      ######################## affichage_POPUP #####################################
      sync()
      num_soud = to_str(num)
      popup1 = "popup Config. : " + type_soud + " n°" + num_soud + " : placer " + etape_soud + " & Valider"             #on ouvre un popup
      socket_open("127.0.0.1", 29999, "internal") # open internal socket
      socket_send_line(popup1, "internal")     #Affichage message
      socket_send_byte(10, "internal")
      sync()
  end
  #-

  def popUp_tropSoudures():
      close_popup()
      popUp_tropSoudures = "Ajout impossible, deja 10 soudures de ce type"
      socket_open("127.0.0.1",29999,"internal") # open internal socket
      socket_send_line(popUp_tropSoudures,"internal")     #Affichage message
      socket_send_byte(10,"internal")
  end
  #-
  $ 41 "Mouvements soudures"
  $ 42 "Script: fcts_balayage.script"
  def fct_determineAxeBalayage(p_start,p_stop):

      global  diff_x = norm(p_start[0]-p_stop[0])
      global  diff_y = norm(p_start[1]-p_stop[1])
      global  diff_z = norm(p_start[2]-p_stop[2])

      global offset_x =  0
      global offset_y =  0
      global offset_z = 0

      local tolerance = 0.02



      if ( (diff_z >0.05) ):
          offset_z = 1
      end

      if ( (diff_x >tolerance) or (offset_z == 1)):
          offset_y = 1
      end

      if ( (diff_y >tolerance) or (offset_z == 1)):
          offset_x = 1
      end

  end

  def fct_set_offset():

      if (offset_x == 1):
          offset[0] = sin((i/cycle_duration)*2.0*pi) * amplitude
      end

      if (offset_y == 1):
          offset[1] = sin((i/cycle_duration)*2.0*pi) * amplitude
      end

  end

  thread runBalayage():
    while (True):
        global ctrl_frequency=350.0
        global weave_frequency=1.2
        global amplitude=0.003
        global cycle_duration=(ctrl_frequency / weave_frequency)
        global pi=3.14159
        global offset=[0.0, 0.0, 0.0, 0.0, 0.0, 0.0]
        global i=0
        path_offset_enable()
        global alpha=0.1
        path_offset_set_alpha_filter(alpha)

        while (True):
          fct_set_offset()
          path_offset_set(offset, 2)
          global i=i+1
          sync()
        end
      end

  end

  def fct_activerBalayage(p_start, p_stop,amplitude, frequence):

      fct_determineAxeBalayage(p_start,p_stop)
      amplitude_thr = amplitude
      frequence_thr = frequence
      global thr_runBalayage = run runBalayage()

  end

  def fct_desactiverBalayage():

      kill thr_runBalayage

  end

  def fct_demande_amplitude():

      amplitude = request_integer_from_primary_client("amplitude du balayage en mm :")
      while (amplitude <=0):
          amplitude = request_integer_from_primary_client("amplitude du balayage en mm :")
      end

      amplitude = amplitude/1000

      return amplitude

  end


  def fct_demande_frequence():

      frequence = request_float_from_primary_client("frequence du balayage en Hz :")
      while (frequence <=0):
          frequence = request_float_from_primary_client("frequence du balayage en Hz :")
      end

      return frequence

  end
  $ 43 "Script: fcts_ralentir_fin_ligne.script"
  def fct_calcul_point_inter(p_debut,p_fin):

      local p_inter = p_fin

      local poucentage = 0.95
      local inc = 0
      local vecteur_global = p[0,0,0,0,0,0]
      local vecteur_reduit = p[0,0,0,0,0,0]

      while (inc < 6):   #a valider avec d'autres tests (peut etre faire une moyenne)
          vecteur_global[inc] = p_fin[inc] - p_debut[inc]
          vecteur_reduit[inc] = vecteur_global[inc]*poucentage
          p_inter[inc] = p_debut[inc] + vecteur_reduit[inc]
          inc = inc +1
      end

      return p_inter
    end


  $ 44 "General"
  $ 45 "Script: diverses.script"
  def attente_carters_ouverts():
      global debug = 2
      # vérifier que les carter sont ouverts,
      # sinon attendre en faisant clignoter les leds

      while ((get_configurable_digital_in(add_SecuGaucheOk) == True) or (get_configurable_digital_in(add_SecuDroiteOK) == True)):

          sync()
          # 94 "'clingottement pour signifier qu'il y  un defaut sur un des carters '"
          set_standard_digital_out(add_Dcy_Voyant, False)
          set_configurable_digital_out(add_Led_Arret, False)
          sleep(0.5)
          set_standard_digital_out(add_Dcy_Voyant, True)
          set_configurable_digital_out(add_Led_Arret, True)
          sleep(0.5)
          sync()
      end

      #carter OK, RAZ des sorties
      set_standard_digital_out(add_Dcy_Voyant, False)
      set_configurable_digital_out(add_Led_Arret, False)
      sleep(2)
      sync()

      global debug = 3

  end
  #-

  def deplacement_depart_init():

      global angle_base = get_actual_joint_positions ()
      if (angle_base[0] <= 0.7):
          if (angle_base[0] >= 1.6):
              # 116 "Départ"        A CHANGER PAR UNE POSTION ENREGISTREE
              movej(pose_depart, a = accelerationHorsSoudure, v = vitesseHorsSoudure)
          else:
              if (angle_base[0] > 1.6):
                  movej(Point_init_D, a = accelerationHorsSoudure, v = vitesseHorsSoudure)
                  movej(Point_avt_initD, a = accelerationHorsSoudure, v = vitesseHorsSoudure)
              else:
                  if (angle_base[0] < 0.7):
                      movej(Point_init_G, a = accelerationHorsSoudure, v = vitesseHorsSoudure)
                  end
              end
          end
      else:
          # 124 "SinonSi angle_base[0]>1.6"
          if (angle_base[0] > 1.6):

              movej(Point_init_D, a = accelerationHorsSoudure, v = vitesseHorsSoudure)
              movej(Point_avt_initD, a = accelerationHorsSoudure, v = vitesseHorsSoudure)
          else:
              if (angle_base[0] < 0.7):
                  movej(Point_init_G, a = accelerationHorsSoudure, v = vitesseHorsSoudure)
              end
          end
      end
      # 131 "Départ"             A CHANGER PAR UNE POSTION ENREGISTREE
      movej(pose_depart, a = accelerationHorsSoudure, v = vitesseHorsSoudure)
      #global angle_base= get_actual_joint_positions ()
      sync()
  end
  #-

  def mode_configuration():
      #nouveau

      if ((config_g == 1) and (config_d == 1)):
          pop_up_config_g_et_d()
      elif ((config_g == 1) and (config_d == 0)):
          pop_up_config_g()
      elif ((config_g == 0) and (config_d == 1)):
          pop_up_config_d()
      elif ((config_g == 0) and (config_d == 0)):
          pop_up_config()
      end

      while ((get_configurable_digital_in(add_ModeExe) == False  ) and (get_standard_digital_in(add_bp_ConfigReglage) == False  )):
          thread Thread_while_145():
              while (True):  # faire clignoter les voyants des tables, pour informer de l'attente d'une action
                  set_standard_digital_out(add_VoyantTableDroite, True)
                  set_standard_digital_out(add_VoyantTableGauche, False)
                  sleep(0.5)
                  set_standard_digital_out(add_VoyantTableDroite, False)
                  set_standard_digital_out(add_VoyantTableGauche, True)
                  sleep(0.5)
                  sync()
              end
          end
          if (get_standard_digital_in(adresse_bp_d) == False and get_standard_digital_in(adresse_bp_g) == False and get_configurable_digital_in(add_ModeExe) == False and get_standard_digital_in(add_bp_ConfigReglage) == False):
              global thread_handler_145 = run Thread_while_145()
              while (get_standard_digital_in(adresse_bp_d) == False and get_standard_digital_in(adresse_bp_g) == False and get_configurable_digital_in(add_ModeExe) == False and get_standard_digital_in(add_bp_ConfigReglage) == False):
                  sync()
              end
              kill thread_handler_145
          end
          if (get_standard_digital_in(adresse_bp_g) == True): #table gauche
              set_standard_digital_out(add_VoyantTableGauche, True)
              set_standard_digital_out(add_VoyantTableDroite, False)
              movej(Point_init_G, a = accelerationHorsSoudure, v = vitesseHorsSoudure, r = 0.006)
              movej(Point_Attente_G, a = accelerationHorsSoudure, v = vitesseHorsSoudure, r = 0.006)
              movej(Point_config_g, a = accelerationHorsSoudure, v = vitesseHorsSoudure)
              global led_cobot = 1
              fun_config_g()
              global led_cobot = 0
              fun_valid_config_g()
              movej(Point_Attente_G, a = accelerationHorsSoudure, v = vitesseHorsSoudure, r = 0.006)
              movej(Point_init_G, a = accelerationHorsSoudure, v = vitesseHorsSoudure, r = 0.006)
              # 170 "Départ"         A CHANGER PAR UNE POSTION ENREGISTREE
              movej(pose_depart, a = accelerationHorsSoudure, v = vitesseHorsSoudure)
          end

          if (get_standard_digital_in(adresse_bp_d) == True): #table droite
              set_standard_digital_out(add_VoyantTableDroite, True)
              set_standard_digital_out(add_VoyantTableGauche, False)
              movej(Point_avt_initD, a = accelerationHorsSoudure, v = vitesseHorsSoudure, r = 0.006)
              movej(Point_init_D, a = accelerationHorsSoudure, v = vitesseHorsSoudure)
              movej(Point_Attente_D, a = accelerationHorsSoudure, v = vitesseHorsSoudure, r = 0.006)
              movej(Point_config_d, a = accelerationHorsSoudure, v = vitesseHorsSoudure)
              global led_cobot = 1
              fun_config_d()
              global led_cobot = 0
              fun_valid_config_d()
              movej(Point_Attente_D, a = accelerationHorsSoudure, v = vitesseHorsSoudure, r = 0.006)
              movej(Point_init_D, a = accelerationHorsSoudure, v = vitesseHorsSoudure, r = 0.006)
              movej(Point_avt_initD, a = accelerationHorsSoudure, v = vitesseHorsSoudure, r = 0.006)
              # 190 "Départ"         A CHANGER PAR UNE POSTION ENREGISTREE
              movej(pose_depart, a = accelerationHorsSoudure, v = vitesseHorsSoudure)
          end
      end

      sync()
  end
  #-

  def mode_Reglage():
      #Pas à Pas
      if ((config_g == 1) and (config_d == 1)):
          pop_up_reg_gd()
          global boucle = 1
      elif ((config_g == 1) and (config_d == 0)):
          pop_up_reg_gd()
          global boucle = 1
      elif ((config_g == 0) and (config_d == 1)):
          pop_up_reg_d()
          global boucle = 1
      else:
          close_popup()
          while (get_standard_digital_in(add_bp_ConfigReglage) == True):
              popup("Aucune configuration n'est actuellement detectée.", "Erreur", False, True, blocking = True)
          end
      end



      global boucle = 1
      while ((get_configurable_digital_in(add_ModeExe) == False  ) and (boucle == 1) and (get_standard_digital_in(add_bp_ConfigReglage) == True  )):
          thread Thread_while_208():
              while (True):
                  if (config_g == 1):
                      set_standard_digital_out(add_VoyantTableGauche, True)
                  end
                  if (config_d == 1):
                      set_standard_digital_out(add_VoyantTableDroite, True)
                  end
                  sleep(0.5)
                  set_standard_digital_out(add_VoyantTableGauche, False)
                  set_standard_digital_out(add_VoyantTableDroite, False)
                  sleep(0.5)
              end
          end
          if (get_standard_digital_in(adresse_bp_d) == False and get_standard_digital_in(adresse_bp_g) == False and get_configurable_digital_in(add_ModeExe) == False and get_standard_digital_in(add_bp_ConfigReglage) == True):
              global thread_handler_208 = run Thread_while_208()
              while (get_standard_digital_in(adresse_bp_d) == False and get_standard_digital_in(adresse_bp_g) == False and get_configurable_digital_in(add_ModeExe) == False and get_standard_digital_in(add_bp_ConfigReglage) == True):
                  sync()
              end
              kill thread_handler_208
          end
          if (get_standard_digital_in(adresse_bp_g) == True): #table gauche
              global safe_mode = 1
              set_standard_digital_out(add_VoyantTableGauche, True)
              set_standard_digital_out(add_VoyantTableDroite, False)
              movej(Point_init_G, a = accelerationHorsSoudure, v = vitesseHorsSoudure, r = 0.006)
              movej(Point_Attente_G, a = accelerationHorsSoudure, v = vitesseHorsSoudure, r = 0.006)
              movej(pose_inter_g, a = accelerationHorsSoudure, v = vitesseHorsSoudure)
              global led_cobot = 1
              fun_Pas_A_Pas_g()
              global led_cobot = 0
              global safe_mode = 0
              global boucle = 0
          end
          if (get_standard_digital_in(adresse_bp_d) == True): #table droite
              global safe_mode = 1
              set_standard_digital_out(add_VoyantTableDroite, True)
              set_standard_digital_out(add_VoyantTableGauche, False)
              movej(Point_avt_initD, a = accelerationHorsSoudure, v = vitesseHorsSoudure, r = 0.006)
              movej(Point_init_D, a = accelerationHorsSoudure, v = vitesseHorsSoudure, r = 0.006)
              movej(pose_inter_d, a = accelerationHorsSoudure, v = vitesseHorsSoudure)
              global led_cobot = 1
              fun_Pas_A_Pas_d()
              global led_cobot = 0
              global safe_mode = 0
              global boucle = 0
          end
      end

      sync()
  end
  #-

  def mode_Execution():

      if ((config_g == 1) and (config_d == 1)):
          pop_up_exe()
          global boucle = 1
      elif ((config_g == 1) and (config_d == 0)):
          pop_up_exe_g()
          global boucle = 1
      elif ((config_g == 0) and (config_d == 1)):
          pop_up_exe_d()
          global boucle = 1
      else:
          close_popup()
          while (get_configurable_digital_in(add_ModeExe) == True):
              popup("Aucune programmation n'est actuellement detectée, veillez à programmer une pièce avant de vouloir l'éxécuter.", "Erreur", False, True, blocking = True)
          end
      end

      while (( get_configurable_digital_in(add_ModeExe) == True  ) and (boucle == 1)):
          thread Thread_while_259():
              while (True):
                  if (config_g == 1):
                      set_standard_digital_out(add_VoyantTableGauche, True)
                  end
                  if (config_d == 1):
                      set_standard_digital_out(add_VoyantTableDroite, True)
                  end
                  sleep(0.5)
                  set_standard_digital_out(add_VoyantTableGauche, False)
                  set_standard_digital_out(add_VoyantTableDroite, False)
                  sleep(0.5)
              end
          end

          if (get_standard_digital_in(adresse_bp_d) == False and get_standard_digital_in(adresse_bp_g) == False and get_configurable_digital_in(add_ModeExe) == True):
              global thread_handler_259 = run Thread_while_259()
              while (get_standard_digital_in(adresse_bp_d) == False and get_standard_digital_in(adresse_bp_g) == False and get_configurable_digital_in(add_ModeExe) == True):
                  sync()
              end
              kill thread_handler_259
          end

          if ((get_standard_digital_in(adresse_bp_g) == True  ) and (config_g == True  )): #table de gauche
              pop_up_deb_exe_g()
              global boucle_g = 1
              while (boucle_g == 1):  #Boucler une fois, tant que la soudure n'est pas finie
                  set_configurable_digital_out(add_CmdCarterBit1, True)#commande la fermeture du carter

                  set_standard_digital_out(add_VoyantTableGauche, True) #commande des voyants
                  set_standard_digital_out(add_VoyantTableDroite, False)
                  sleep(0.25)
                  set_standard_digital_out(add_VoyantTableGauche, False)
                  sleep(0.25)

                  if (get_configurable_digital_in(add_SecuGaucheOk) == False): #si les carter ne sont pas en position : voyant et attente
                      set_standard_digital_out(add_VoyantTableGauche, True)
                      while (get_configurable_digital_in(add_SecuGaucheOk) == False):
                          sync()
                      end
                  end

                  if (get_configurable_digital_in(add_SecuGaucheOk) == True): # attente de la confirmation de la position du carter -> début soudure
                      global secu_g = 1
                      set_standard_digital_out(add_VoyantTableGauche, True)
                      movej(Point_init_G, a = accelerationHorsSoudure, v = vitesseHorsSoudure, r = 0.006)
                      fun_execution_g()
                      movej(Point_Attente_G, a = accelerationHorsSoudure, v = vitesseHorsSoudure, r = 0.006)
                      movej(Point_init_G, a = accelerationHorsSoudure, v = vitesseHorsSoudure, r = 0.006)
                      # 294 "Départ"         A CHANGER PAR UNE POSTION ENREGISTREE
                      movej(pose_depart, a = accelerationHorsSoudure, v = vitesseHorsSoudure)
                      set_configurable_digital_out(add_CmdCarterBit1, False)
                      global secu_g = 0
                      global boucle_g = 0
                  end
              end
              global boucle = 0
          else:
              if ((get_standard_digital_in(adresse_bp_g) == True  ) and (config_g == False  )): # si la table n'est pas enregistrée comme configurée
                  close_popup()
                  popup("Aucune programmation n'est actuellement detectée sur la table gauche, veillez à programmer une pièce avant de vouloir l'éxécuter.", "Erreur", False, True, blocking = True)
                  global boucle = 0
              end
          end
          if ((get_standard_digital_in(adresse_bp_d) == True  ) and (config_d == True  )):  #table de droite
              global boucle_d = 1
              pop_up_deb_exe_d()
              while (boucle_d == 1):  #Boucler une fois, tant que la soudure n'est pas finie
                  set_configurable_digital_out(add_CmdCarterBit2, True) #commande la fermeture du carter

                  set_standard_digital_out(add_VoyantTableGauche, False)#commande des voyants
                  set_standard_digital_out(add_VoyantTableDroite, True)
                  sleep(0.25)
                  set_standard_digital_out(add_VoyantTableDroite, False)
                  sleep(0.25)

                  if (get_configurable_digital_in(add_SecuDroiteOK) == False): #si les carter ne sont pas en position : voyant et attente
                      set_standard_digital_out(add_VoyantTableDroite, True)
                      while (get_configurable_digital_in(add_SecuDroiteOK) == False):
                          sync()
                      end
                  end

                  if (get_configurable_digital_in(add_SecuDroiteOK) == True):# attente de la confirmation de la position du carter -> début soudure
                      global secu_d = 1
                      set_standard_digital_out(add_VoyantTableDroite, True)
                      movej(Point_avt_initD, a = accelerationHorsSoudure, v = vitesseHorsSoudure)
                      fun_execution_d()
                      set_configurable_digital_out(add_CmdCarterBit2, False)
                      global secu_d = 0
                      global boucle_d = 0
                  end
              end
              global boucle = 0
          else:
              if ((get_standard_digital_in(adresse_bp_d) == True  ) and (config_d == False  )): # si la table n'est pas enregistrée comme configurée
                  close_popup()
                  popup("Aucune programmation n'est actuellement detectée sur la table droite, veillez à programmer une pièce avant de vouloir l'éxécuter.", "Erreur", False, True, blocking = True)
                  global boucle = 0
              end
          end
      end
      sync()
  end
  #-
  $ 46 "Script: general.script"
  def General():

      while (True):

          global debug = 1
          #INTIALISATION
          safe_mode = 0
          set_configurable_digital_out(add_CmdCarterBit1, False) #stop commande carter
          set_configurable_digital_out(add_CmdCarterBit2, False)

          attente_carters_ouverts() #éviter un contact avec le bras

          deplacement_depart_init() #premier déplacement à gérer en focntion de la position réel du robot lors de l'init

          # TEST DES MODES :
          # lecture de la postion des Bps
          if ((get_configurable_digital_in(add_ModeExe) == False) and (get_standard_digital_in(add_bp_ConfigReglage) == False)):
              mode_configuration()#l 55-> 127
          elif ((get_configurable_digital_in(add_ModeExe) == False) and (get_standard_digital_in(add_bp_ConfigReglage) == True  )):
              mode_Reglage() #l 127 -> 199
          elif (get_configurable_digital_in(add_ModeExe) == True):
              mode_Execution() #
          else:
              #faire erreur
          end
      end

  end
  $ 76 "Thread_1"
  thread Thread_1():
    while (True):
      $ 77 "Test_Ordre_Marche"
      $ 78 "If Test_Ordre_Mar≟ True "
      if (Test_Ordre_Mar ==   True  ):
        $ 79 "If config_d ≟ 1  or  config_g ≟ 1"
        if (config_d  ==  1   or   config_g  ==  1):
          $ 80 "Set Ordre_Marche=On"
          set_standard_digital_out(0, True)
          $ 81 "Wait: 0.5"
          sleep(0.5)
          $ 82 "If Reponse_Ordre≟ False "
          if (get_standard_digital_in(4) ==   False  ):
            $ 83 "'Si aucune reponse n'a etait recue, arret du programme'"
            # 'Si aucune reponse n'a etait recue, arret du programme'
            $ 84 "close_popup()"
            close_popup()
            $ 85 "Popup: Defaut : L'Ordre marche a ete coupe ( le poste est peu-etre eteint ) "
            popup("Defaut : L'Ordre marche a ete coupe ( le poste est peu-etre eteint ) ", "Error", False, True, blocking=False)
            halt
          end
          $ 86 "Test_Ordre_Mar≔ False "
          global Test_Ordre_Mar=  False
          $ 87 "sync()"
          sync()
        end
      end
      $ 88 "Erreur ordre marche pendant utilisation"
      $ 89 "If Arc_On≟ True   and Reponse_Arc≟ True  and Reponse_Ordre≟ False "
      if (get_standard_digital_out(1) ==   True     and  get_standard_digital_in(5) ==   True    and  get_standard_digital_in(4) ==   False  ):
        $ 90 "'Test pour savoir si ordre marche a ete coupe pendant utilisation'"
        # 'Test pour savoir si ordre marche a ete coupe pendant utilisation'
        $ 91 "close_popup()"
        close_popup()
        $ 92 "Popup: Defaut : Mise sous puissance coupee pendant la trajectoire"
        popup("Defaut : Mise sous puissance coupee pendant la trajectoire", "Error", False, True, blocking=False)
        halt
      end
      $ 93 "sync()"
      sync()
    end
  end
  threadId_Thread_1 = run Thread_1()
  $ 94 "Thread_2"
  thread Thread_2():
    while (True):
      $ 95 "mode_soudure"
      $ 96 "If Mode_soudure ≟  True "
      if (get_configurable_digital_in(3)  ==    True  ):
        $ 97 "If Mode_soudure≟ True  and soudure_on ≟ True "
        if (get_configurable_digital_in(3) ==   True    and  soudure_on  ==   True  ):
          $ 98 "fin_soud≔0"
          global fin_soud=0
          $ 99 "Test_Ordre_Mar≔ True "
          global Test_Ordre_Mar=  True
          $ 100 "Test_Job≔ True "
          global Test_Job=  True
          $ 101 "Wait Test_Ordre_Mar≟ False "
          while (not(Test_Ordre_Mar ==   False  )):
            sync()
          end
          $ 102 "Wait Test_Job≟ False "
          while (not(Test_Job ==   False  )):
            sync()
          end
          $ 103 "Set Arc_On=On"
          set_standard_digital_out(1, True)
          $ 104 "Test_Gaz≔ True "
          global Test_Gaz=  True
          $ 105 "'Test_Gaz permet de faire un appel dans le thread pour tester l'arriver gaz'"
          # 'Test_Gaz permet de faire un appel dans le thread pour tester l'arriver gaz'
          $ 106 "Wait Valide_Gaz≟ True "
          while (not(Valide_Gaz ==   True  )):
            sync()
          end
          $ 107 "'Valide_Gaz permet  de connaitre quand le traitement de l'arriver gaz est terminer ans le thread.'"
          # 'Valide_Gaz permet  de connaitre quand le traitement de l'arriver gaz est terminer ans le thread.'
        else:
          $ 108 "ElseIf Mode_soudure ≟ True  and soudure_on ≟ False "
          if (get_configurable_digital_in(3)  ==   True    and  soudure_on  ==   False  ):
            $ 109 "'Attente post debit gaz'"
            # 'Attente post debit gaz'
            $ 110 "Set Arc_On=Off"
            set_standard_digital_out(1, False)
            $ 111 "Test_Gaz≔ False "
            global Test_Gaz=  False
            $ 112 "Loop Reponse_Arc ≟ 1"
            while (get_standard_digital_in(5)  ==  1):
              $ 113 "fin_soud≔0"
              global fin_soud=0
              $ 114 "sync()"
              sync()
            end
            $ 115 "fin_soud≔1"
            global fin_soud=1
          end
        end
      end
      $ 116 "sync()"
      sync()
    end
  end
  threadId_Thread_2 = run Thread_2()
  $ 117 "Thread_3"
  thread Thread_3():
    while (True):
      $ 118 "led_cobot_2"
      $ 119 "If led_cobot ≟ True "
      if (led_cobot  ==   True  ):
        $ 120 "If valider_bp_co ≟ True "
        if (get_tool_digital_in(0)  ==   True  ):
          $ 121 "Loop 3 times"
          Loop_4 = 0
          while (Loop_4 < 3):
            $ 122 "Set TO[1]=On"
            set_tool_digital_out(1, True)
            $ 123 "Wait: 0.25"
            sleep(0.25)
            $ 124 "Set TO[1]=Off"
            set_tool_digital_out(1, False)
            $ 125 "Wait: 0.25"
            sleep(0.25)
            $ 126 "sync()"
            sync()
            Loop_4 = Loop_4 + 1
          end
        end
        $ 127 "sync()"
        sync()
      end
      $ 128 "sync()"
      sync()
      $ 129 "sync()"
      sync()
    end
  end
  threadId_Thread_3 = run Thread_3()
  $ 130 "Thread_4"
  thread Thread_4():
    while (True):
      $ 131 "led_cobot"
      $ 132 "If led_cobot ≟ True "
      if (led_cobot  ==   True  ):
        $ 133 "Loop led_cobot ≟  True "
        while (led_cobot  ==    True  ):
          $ 134 "Set TO[0]=On"
          set_tool_digital_out(0, True)
          $ 135 "Wait: 0.5"
          sleep(0.5)
          $ 136 "Set TO[0]=Off"
          set_tool_digital_out(0, False)
          $ 137 "Wait: 0.5"
          sleep(0.5)
          $ 138 "sync()"
          sync()
        end
        $ 139 "sync()"
        sync()
      else:
        $ 140 "Else" "noBreak"
        $ 141 "Set TO[0]=Off"
        set_tool_digital_out(0, False)
        $ 142 "Set TO[1]=Off"
        set_tool_digital_out(1, False)
      end
      $ 143 "sync()"
      sync()
    end
  end
  threadId_Thread_4 = run Thread_4()
  $ 144 "Thread_5"
  thread Thread_5():
    while (True):
      $ 145 "Test_Arc_On"
      $ 146 "Erreur gaz pendant utilisation"
      $ 147 "Timer_gaz"
      $ 148 "If Test_Gaz≟ True "
      if (Test_Gaz ==   True  ):
        $ 149 "Wait: 1.0"
        sleep(1.0)
        $ 150 "Loop Reponse_Arc≟ False  and Arc_On≟ True "
        thread Thread_while_150():
          while (True):
            $ 151 "'La boucle permet d'activer le timer et tester deux condition pour les Defaults'"
            # 'La boucle permet d'activer le timer et tester deux condition pour les Defaults'
            $ 152 "timer_ret_gaz: Start"
            timer_ret_gaz_is_counting = True
            $ 153 "If timer_ret_gaz>0.5"
            global thread_flag_153=0
            thread Thread_if_153():
              $ 154 "'Le timer permet de realiser une attente '"
              # 'Le timer permet de realiser une attente '
              $ 155 "close_popup()"
              close_popup()
              $ 156 "Popup: Defaut : Pas de retour flux, stabilisation gaz"
              popup("Defaut : Pas de retour flux, stabilisation gaz", "Error", False, True, blocking=False)
              halt
              $ 157 "sync()"
              sync()
              thread_flag_153 = 1
            end
            if (timer_ret_gaz>0.5):
              global thread_handler_153=run Thread_if_153()
              while (thread_flag_153 == 0):
                if not(timer_ret_gaz>0.5):
                  kill thread_handler_153
                  thread_flag_153 = 2
                else:
                  sync()
                end
              end
            else:
              thread_flag_153 = 2
            end
            if (thread_flag_153 == 2):
              $ 158 "ElseIf Reponse_Ordre≟ False "
              if (get_standard_digital_in(4) ==   False  ):
                $ 159 "'Cette condition nous permet de pouvoir tout couper ordre marche pendant la boucle.'"
                # 'Cette condition nous permet de pouvoir tout couper ordre marche pendant la boucle.'
                $ 160 "close_popup()"
                close_popup()
                $ 161 "Popup: Defaut : Perte retour de signal, mise sous puissance generateur"
                popup("Defaut : Perte retour de signal, mise sous puissance generateur", "Error", False, True, blocking=False)
                halt
                $ 162 "sync()"
                sync()
              end
            end
          end
        end
        if (get_standard_digital_in(5) ==   False    and  get_standard_digital_out(1) ==   True  ):
          global thread_handler_150=run Thread_while_150()
          while (get_standard_digital_in(5) ==   False    and  get_standard_digital_out(1) ==   True  ):
            sync()
          end
          kill thread_handler_150
        end
        $ 163 "Valide_Gaz≔ True "
        global Valide_Gaz=  True
        $ 164 "timer_ret_gaz: Reset"
        timer_ret_gaz = 0
        $ 165 "sync()"
        sync()
      end
      $ 166 "sync()"
      sync()
    end
  end
  threadId_Thread_5 = run Thread_5()
  $ 175 "Thread_7"
  thread Thread_7():
    while (True):
      $ 176 "secu"
      $ 177 "If SecuGaucheOk ≟  False  and secu_g ≟ 1"
      if (get_configurable_digital_in(4)  ==    False    and  secu_g  ==  1):
        $ 178 "close_popup()"
        close_popup()
        $ 179 "Popup: ATTENTION : Defaut carter !"
        popup("ATTENTION : Defaut carter !", "Error", False, True, blocking=False)
        halt
      else:
        $ 180 "ElseIf SecuDroiteOk ≟ False  and secu_d ≟ 1"
        if (get_configurable_digital_in(5)  ==   False    and  secu_d  ==  1):
          $ 181 "close_popup()"
          close_popup()
          $ 182 "Popup: ATTENTION : Defaut carter !"
          popup("ATTENTION : Defaut carter !", "Error", False, True, blocking=False)
          halt
        end
      end
      $ 183 "sync()"
      sync()
    end
  end
  threadId_Thread_7 = run Thread_7()
  $ 184 "Thread_8"
  thread Thread_8():
    while (True):
      $ 185 "bloq_soud_arret"
      $ 186 "If Mode_soudure≟ False  and Test_Gaz ≟ True "
      if (get_configurable_digital_in(3) ==   False    and  Test_Gaz  ==   True  ):
        $ 187 "close_popup()"
        close_popup()
        $ 188 "Popup: Defaut : L'ordre de soudure a ete coupe pendant l'utilisation."
        popup("Defaut : L'ordre de soudure a ete coupe pendant l'utilisation.", "Error", False, True, blocking=False)
        halt
        $ 189 "sync()"
        sync()
      end
      $ 196 "sync()"
      sync()
    end
  end
  threadId_Thread_8 = run Thread_8()
  $ 207 "Thread_10"
  thread Thread_10():
    while (True):
      $ 208 "reglage"
      $ 209 "If safe_mode ≟ 1  and Mode_Exe ≟  True "
      if (safe_mode  ==  1   and  get_configurable_digital_in(7)  ==    True  ):
        $ 210 "close_popup()"
        close_popup()
        $ 211 "Popup: STOP !!!!"
        popup("STOP !!!!", "Error", False, True, blocking=False)
        halt
      end
      $ 212 "sync()"
      sync()
      $ 213 "sync()"
      sync()
    end
  end
  threadId_Thread_10 = run Thread_10()
  $ 47 "Robot Program"
  $ 48 "General()"
  General()
end
